(* CODESYS project Trafficlight_DAN_2.project

Project tree, tasks and I/O mapping:
  Device : CODESYS Control Win V3, 3S - Smart Software Solutions GmbH, order no. 305021, version 3.5.10.30
    application Application
      libraries: Standard, * (System)
      task MainTask (cyclic, interval t#20ms, priority 1) calls PLC_PRG
      task VISU_TASK (cyclic, interval 100 ms, priority 31) calls VisuElems.Visu_Prg
      program PLC_PRG [FBD]
      function block Normal_Cycle_FB [ST]
      visualisation Visualization
  text list GlobalTextList
*)

// Device/Application/PLC_PRG
PROGRAM PLC_PRG
VAR
	Switch_general_enable : BOOL := FALSE;
	Time_red : INT :=5;
	Time_yellow : INT :=5;
	Time_green : INT :=5;
	Led_red : BOOL :=FALSE;
	Led_yellow : BOOL :=FALSE;
	Led_green : BOOL :=FALSE;
	Switch_Enable_blink : BOOL :=FALSE; 
	Normal_cycle: Normal_Cycle_FB;
END_VAR

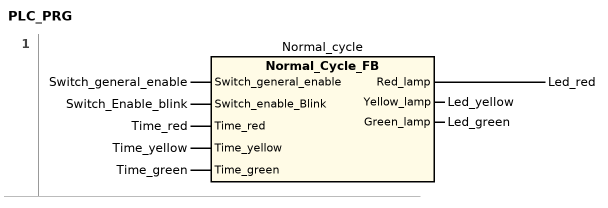
// NETWORK 1
Normal_cycle(
    Switch_general_enable := Switch_general_enable,
    Switch_enable_Blink := Switch_Enable_blink,
    Time_red := Time_red,
    Time_yellow := Time_yellow,
    Time_green := Time_green,
    Yellow_lamp => Led_yellow,
    Green_lamp => Led_green); // Normal_Cycle_FB
Led_red := Normal_cycle.Red_lamp;

END_PROGRAM

// Device/Application/Normal_Cycle_FB
FUNCTION_BLOCK Normal_Cycle_FB
VAR_INPUT
	Switch_general_enable : BOOL := FALSE;
	Switch_enable_Blink : BOOL := FALSE;
	Time_red : INT := 0;
	Time_yellow : INT := 0;
	Time_green : INT := 0;
	END_VAR
	
VAR_OUTPUT
	Red_lamp : BOOL :=FALSE;
	Yellow_lamp : BOOL :=FALSE;
	Green_lamp : BOOL :=FALSE;
END_VAR

VAR
	State_Trafficlight : INT := 0;
	Set_ON_red : BOOL := FALSE;
	Set_ON_yellow : BOOL := FALSE;
	Set_ON_green : BOOL := FALSE;
	Clock_red : TON;
	Clock_yellow : TON;
	Clock_green : TON;
	Count_red : INT :=0;
	Count_yellow : INT :=0;
	Count_green : INT :=0;
	SWITCH: INT;
END_VAR

IF Switch_general_enable = TRUE THEN
	IF State_Trafficlight = 0 THEN
		State_Trafficlight := 1;
	END_IF
	CASE (State_Trafficlight) OF
		1:
		Red_lamp := TRUE;
		Clock_red(IN:=TRUE, PT:=T#1S);
		IF NOT(Clock_red.Q) THEN
			RETURN;
		END_IF
		Clock_red(IN:=FALSE);
		Count_red := Count_red +1;
		IF Count_red = Time_red THEN
			State_Trafficlight := 2;
			Red_lamp := FALSE;
			Count_red :=0;
		END_IF
		
		2:
		Green_lamp := TRUE;
		Clock_green(IN:=TRUE, PT:=T#1S);
		IF NOT(Clock_green.Q) THEN
			RETURN;
		END_IF
		Clock_green(IN:=FALSE);
		Count_green := Count_green +1;
		IF Count_green = Time_green THEN
			State_Trafficlight := 3;
			Green_lamp := FALSE;
			Count_green :=0;
		END_IF
		
		3:
		Green_lamp := TRUE;
		Yellow_lamp :=TRUE;
		Clock_yellow(IN:=TRUE,PT:=T#1S);
		IF NOT(Clock_yellow.Q) THEN
			RETURN;
		END_IF
		Clock_yellow(IN:=FALSE);
		Count_yellow := Count_yellow +1;
		IF Count_yellow = Time_yellow THEN
			State_Trafficlight := 1;
			Green_lamp := FALSE;
			Yellow_lamp :=FALSE;
			Count_yellow :=0;
		END_IF
			
	END_CASE
	
ELSE
	Red_lamp := FALSE;
	Yellow_lamp := FALSE;
	Green_lamp := FALSE;
	State_Trafficlight := 0;
	Count_red :=0;
	Count_yellow :=0;
	Count_green :=0;
END_IF

END_FUNCTION_BLOCK

// Device/Application/Visualization
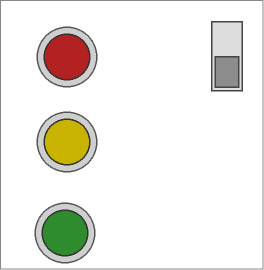
VISUALIZATION Visualization  // 264x270
    Lamp1 (32,107 70x70), variable: PLC_PRG.Led_yellow, style: Lamp-Lamp1-Yellow
    Lamp1 (32,22 70x70), variable: PLC_PRG.Led_red, style: Lamp-Lamp1-Red
    Lamp1 (30,198 70x70), variable: PLC_PRG.Led_green, style: Lamp-Lamp1-Green
    DipSwitch (192,21 70x70), variable: PLC_PRG.Switch_general_enable, behaviour: TOGGLE, style: Switch-DipSwitch-Gray
END_VISUALIZATION
